# EPICS autosave request: iocBoot/sioc-li24-bl01/blen_manual.req
file "manual.req" AREA=LI24,POS=887,INST=BL21A
file "manual.req" AREA=LI24,POS=887,INST=BL21B
